// TIA Portal V17 export
// export: Created 2024-09-02T12:50:37.7193319Z, ExportSetting WithDefaults, DisplayName Totally Integrated Automation Portal, DisplayVersion V17, DisplayName TIA Portal Openness, DisplayVersion V17, DisplayName TIA Portal Version Control Interface, DisplayVersion V17, DisplayName STEP 7 Professional, DisplayVersion V17, DisplayName STEP 7 Safety, DisplayVersion V17, DisplayName WinCC Professional, DisplayVersion V17
TYPE "OP40"
// stored: IsFailsafeCompliant false
   STRUCT
      "Data for Proces" : Struct
         "Proces Selected" : Array[1..8] of Bool;
         reserve : Array[0..1] of Byte;
      END_STRUCT;
      Status_Station : Struct
         Operation_Status : Struct
            "Proces #1" { S7_SetPoint := 'True'} : "Proces_r";
            "Proces #2" { S7_SetPoint := 'True'} : "Proces_r";
            "Proces #3" { S7_SetPoint := 'True'} : "Proces_r";
            "Proces #4" { S7_SetPoint := 'True'} : "Proces_r";
            "Proces #5" { S7_SetPoint := 'True'} : "Proces_r";
            "Proces #6" { S7_SetPoint := 'True'} : "Proces_r";
            "Proces #7" { S7_SetPoint := 'True'} : "Proces_r";
            "Proces #8" { S7_SetPoint := 'True'} : "Proces_r";
         END_STRUCT;
      END_STRUCT;
      Restult_Data : Struct
         "Press DA solenoids 1" { S7_SetPoint := 'True'} : "Pressing_R";
         "Press DA solenoids 2" { S7_SetPoint := 'True'} : "Pressing_R";
         "Press DA solenoids 3" { S7_SetPoint := 'True'} : "Pressing_R";
         "Scan DA solenoids 1" { S7_SetPoint := 'True'} : "DMC_Solenoid";
         "Scan DA solenoids 2" { S7_SetPoint := 'True'} : "DMC_Solenoid";
         "Scan DA solenoids 3" { S7_SetPoint := 'True'} : "DMC_Solenoid";
         Reserve : Array[1..2] of Byte;
      END_STRUCT;
      Worker_ID { S7_SetPoint := 'True'} : "typ_Key";
      Reserve : Array[0..18] of Byte;
   END_STRUCT;
END_TYPE
